FUNCTION F_ComputeLengthSize : UDINT
VAR_INPUT
    nLength : UDINT;
END_VAR


F_ComputeLengthSize := F_ComputeRawVarint32Size(nLength);

END_FUNCTION

(* stored: Version 1.1.0.1
   POU F_ComputeLengthSize: Id {c5dda08b-777e-49c6-908f-0d57124e6764}, SpecialFunc None *)
